FUNCTION Convert_DINT_TO_ULINT : Hresult
VAR_INPUT
	in : DINT;
	out : REFERENCE TO ULINT;
END_VAR
VAR
	converted : ULINT;
END_VAR
VAR CONSTANT
	INCOMPATIBLE : HRESULT := 16#9811070E;
END_VAR

converted := DINT_TO_ULINT(in);

IF (ULINT_TO_DINT(converted) <> in) THEN
	Convert_DINT_TO_ULINT := INCOMPATIBLE;
	RETURN;
END_IF

out := converted;

END_FUNCTION

(* stored: Version 1.1.0.1, ProductVersion 3.1.4024.12
   POU Convert_DINT_TO_ULINT: Id {dcbb3c0e-fd8a-475a-ad00-65d0df3a5ac9}, SpecialFunc None *)
